{attribute addProperty BoxType "EL4712--0000"}
{attribute addProperty Id "Ch2_CycleCountAT %Q*UINT162"}
{attribute addProperty CRC "3950150844"}
{attribute addProperty SizeInBites "16"}
{attribute addProperty SizeInBytes "2"}
TYPE Ch2_CycleCount_EB7284BC :
STRUCT
	{attribute addProperty Name "Ch2_CycleCount"}
	Ch2_CycleCount AT %Q* : UINT;
END_STRUCT
END_TYPE

(* stored: Version 1.2.0.0, ProductVersion 3.1.4024.9
   DUT Ch2_CycleCount_EB7284BC: Id {5b8332ac-766d-420e-a725-7f9cf429ce94} *)
